PROGRAM MAIN
VAR


END_VAR

(*Kalla på IOs*)
F15_AS3_AI();

(*Kalla på program*)

F15_ClusterCtrl();
F15_ClusterCtrl_Larm();


PLC_Batteri_Larm();
MAIN_loggning();

(*Kalla på Systemprogram*)
PersistentData();
PLC_TID();
WatchDog_PLC();

END_PROGRAM

(* stored: Version 1.1.0.1, ProductVersion 3.1.4022.3
   POU MAIN: Id {c9d8b898-8938-4f73-b698-bd45bf9b5389}, SpecialFunc None *)
